# EPICS IOC start-up script: urRobotApp/iocsh/paths.iocsh
#- ###################################################################
#- PREFIX     - IOC Prefix
#- N_WP       - (Optional) Number of waypoints (of both types) to load
#- N_ACTIONS  - (Optional) Number of waypoints actions to load
#- N_PATH     - (Optional) Number of paths to load
#- N_PATH_WP  - (Optional) Number of waypoints per path
#- CTRL_PORT  - (Optional) Name of the asyn port for control interface
#- ###################################################################

# Load waypoint and path databases
luash("$(URROBOT)/urRobotApp/iocsh/load_waypoints.lua", "P=$(PREFIX),N=$(N_WP=30)")
luash("$(URROBOT)/urRobotApp/iocsh/load_actions.lua", "P=$(PREFIX),N=$(N_ACTIONS=10)")
luash("$(URROBOT)/urRobotApp/iocsh/load_paths.lua", "P=$(PREFIX),N=$(N_PATH=10),K=$(N_PATH_WP=30),CTRL_PORT=$(CTRL_PORT=rtde_ctrl)")

# Functionality to edit sseq records for waypoint actions
dbLoadRecords("$(CALC)/db/editSseq.db", "P=$(PREFIX),Q=ActionES:")
doAfterIocInit("seq &editSseq, 'P=$(PREFIX),Q=ActionES:'")
